TYPE MODBUS_DATA_MAP :
STRUCT
	_ipAddress : STRING;
	_startAddress : WORD;
END_STRUCT
END_TYPE

(* stored: Version 1.1.0.1, ProductVersion 3.1.0.38
   DUT MODBUS_DATA_MAP: Id {0f7a0a22-8f1c-4cd5-bf22-578fc121e6c0} *)
